(* PLC project SafeLOGIC-1, BrAutomation SafeDESIGNER  4.3.3.7 *)
(* stored: companyURL http://www.br-automation.com, creationDateTime Sat Nov 03 20:50:21 2018 *)

PROGRAM ReleaseOutput

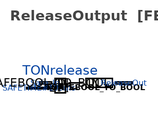
(* FBD diagram, written out as Structured Text *)
TONrelease(IN := Safe_In, PT := SAFETIME#100ms);
ReleaseOut := SAFEBOOL_TO_BOOL(TONrelease.Q);
END_PROGRAM
